{attribute 'linkalways'} 
{attribute 'no_explicit_call' := 'This FB is a CLASS and must be accessed using methods or properties'}
{attribute 'enable_dynamic_creation'}
FUNCTION_BLOCK Node_F_VN_InsertIntoContainer_TcVnVector2_SINT EXTENDS VisionNode
VAR
    aElement : _TcVnVector2_SINT;
    ipContainer : _ITcVnContainer;
    nIndex : _ULINT(0);
    hrPrev : _HRESULT(S_OK);
    hresult : _HRESULT(S_OK);
END_VAR

METHOD PUBLIC  Clone : I_Node
VAR
	pNode : POINTER TO Node_F_VN_InsertIntoContainer_TcVnVector2_SINT;
END_VAR
pNode := __NEW(Node_F_VN_InsertIntoContainer_TcVnVector2_SINT);
Clone := pNode^;
END_METHOD

METHOD FB_init : BOOL
VAR_INPUT
	bInitRetains : BOOL; // if TRUE, the retain variables are initialized (warm start / cold start)
	bInCopyCode : BOOL;  // if TRUE, the instance afterwards gets moved into the copy code (online change)
END_VAR
AddInput('aElement', aElement);
AddInput('ipContainer', ipContainer);
AddInput('nIndex', nIndex);
AddInput('hrPrev', hrPrev);
AddOutput('ipContainer', ipContainer);
AddOutput('hresult',hresult);
END_METHOD

METHOD PROTECTED OnExecute : HRESULT
hresult.Value := F_VN_InsertIntoContainer_TcVnVector2_SINT(
    aElement := aElement.Value,
    ipContainer := ipContainer.Value,
    nIndex := nIndex.Value,
    hrPrev:= hrPrev.Value);
END_METHOD

METHOD PUBLIC PreExecutionCheck
VAR_INPUT
	Check : I_PreExecutionChecks;
END_VAR
Check.IsTrue(ipContainer.IsValid, 'ipContainer must be a valid container');
END_METHOD

END_FUNCTION_BLOCK

(* stored: Version 1.1.0.1, ProductVersion 3.1.4024.13
   POU Node_F_VN_InsertIntoContainer_TcVnVector2_SINT: Id {ad67ee24-3a9f-4454-9a5d-69a19ade5583}, SpecialFunc None
   Folder Constructor: Id {96305d58-dd25-445c-8fe9-0447c1b65fd3}
   Method Clone: Id {dc0e532f-c36e-421c-b477-d1eaa8166a1e}
   Method FB_init: Id {16a84273-c97c-46c4-9cec-2bcf155cceff}
   Method OnExecute: Id {38e10fde-80b6-4e76-a0f8-baf88e7b4d2d}
   Method PreExecutionCheck: Id {a9984799-f45e-4b6e-9d45-742123445845} *)
